PROGRAM MAIN
VAR
	(*	In USA/UK the CSV field separator is a comma.
	In Germany and some other European countries the CSV field separator is a semicolon. *)
	bChangeSeparatorToComma	: BOOL := TRUE;
END_VAR

IF bChangeSeparatorToComma THEN
	DEFAULT_CSV_FIELD_SEP := 16#2C;(* Comma ASCII code *)
ELSE
	DEFAULT_CSV_FIELD_SEP := 16#3B;(* Semicolon ASCII code *)
END_IF

// CSV Sample programs. 
// Open each of the programs and trigger their execution using the bWrite or bRead variables.

P_TextModeWrite();(* This sample program opens and writes CSV file in text mode *)
P_TextModeRead();(* This sample program opens and reads CSV file in text mode *)


// Helper functions.
P_ArgToConvExample();(* This sample program shows the usage of the ARG_TO_CSVFIELD and CSVFILED_TO_ARG conversion functions *)
P_StringToConvExample();(* This sample program shows the usage of the STRING_TO_CSVFIELD and CSVFIELD_TO_STRING conversion functions *)

END_PROGRAM

(* stored: Version 1.1.0.1, ProductVersion 3.1.4024.3
   POU MAIN: Id {6ead28b2-01fa-4be4-a5c6-5ca9fe356e6c}, SpecialFunc None *)
